Staubli VAL3: questionDialog.pgx

public program questionDialog(string x_sMsg (dimensions=1), string& x_sButton[] (dimensions=1), num& x_nResult[] (dimensions=1))
  local bool lExit
  local num nLine
  local num i
  local num nStartLine
  local string l_sMessage
begin
  //---------------------------------
  //      D I A L O G    B O X
  //---------------------------------
  //
  // Show one dialog box. with an confirm question
  //

  if watch(bShowDialog==false,2)==false
    bShowDialog=false
    logMsg("error dialog resoursing")
    return
  else
    setMutex(bShowDialog)
    //call listempty()
    //
    //
    if x_sMsg!=""
      call stringCopy(x_sMsg,sMessage)
      call divideString(sMessage,nLine)
      nStartLine=round(5-nLine/2)
      // Start LINE
      call type(0,nStartLine-2,"┌──────────────────────────────────────┐")
      call type(0,nStartLine-1,"│                                      │")
      // write the message
      for i=0 to nLine
        l_sMessage=sMessage[i]
        call typeCenter(i+nStartLine,l_sMessage,38,false)
        call type(0,nStartLine+i,"│"+l_sMessage+"│")
      endFor
      // end LINE
      call type(0,nStartLine+nLine+1,"│                                      │")
      call type(0,nStartLine+nLine+2,"└──────────────────────────────────────┘")
    endIf
    // write the button message
    call clear(0,13)
    for i=0 to size(x_sButton)-1
      call typeMenu(8-i,x_sButton[i])
    endFor
    lExit=false
    x_nResult=-100
    do
      nKey=get()
      switch (nKey)
        case 270
          x_nResult=0
        break
        case 255
          x_nResult=-1
          bUseEscape=true
        break
        default
          // look if the button press is defined
          if (nKey>=271 and nKey<=278) and ((279-nKey)<=size(x_sButton))
            if x_sButton[278-nKey]!=""
              x_nResult=279-nKey
            endIf
          endIf
        break
      endSwitch
      delay(0)
    until (x_nResult!=-100)
    //
    call nullKey(nKey)
    //
    // release
    bShowDialog=false
    bUseRefresh=true
  endIf
end
